Fanuc KAREL source: ACOS.kl

PROGRAM T
%NOLOCKGROUP
VAR
 v0 : REAL
 res : REAL
BEGIN
 res = ACOS(v0)
END T
